(* LS Electric XG5000 project: 241008_연습문제7 *)
(* PLC LSPLC *)

PROGRAM NewProgram (* task: 스캔 프로그램 *)
VAR
    P0 AT %IX0.0.0 : BOOL;
    P10 AT %QX0.1.0 : BOOL;
    TO : TON;
END_VAR

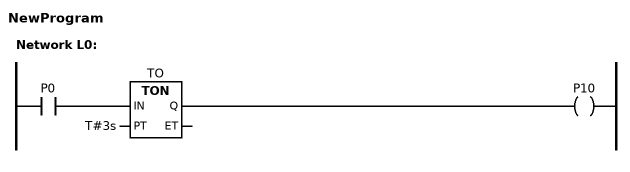
(* Rung L0 *)
TO(IN := P0, PT := T#3s);
P10 := TO.Q;
END_PROGRAM